PROGRAM MAIN
VAR
	_Ivana : BOOL;
END_VAR

END_PROGRAM

(* stored: Version 1.1.0.1, ProductVersion 3.1.4024.12
   POU MAIN: Id {74e2491b-a3cc-4ec7-a1e6-e30b96f03582}, SpecialFunc None *)
